// TIA Portal V17 export
// export: Created 2022-07-20T06:59:51.1083772Z, ExportSetting WithDefaults, DisplayName Totally Integrated Automation Portal, DisplayVersion V17, DisplayName TIA Portal Openness, DisplayVersion V17, DisplayName TIA Portal Version Control Interface, DisplayVersion V17, DisplayName SINAMICS Startdrive Advanced, DisplayVersion V17, DisplayName SINAMICS Startdrive G130, G150, S120, S150, SINAMICS MV, S210, DisplayVersion V17, DisplayName SINAMICS Startdrive G110M, G120, G120C, G120D, G120P, G115D, DisplayVersion V17, DisplayName STEP 7 Professional, DisplayVersion V17, DisplayName STEP 7 Safety, DisplayVersion V17, DisplayName WinCC Advanced, DisplayVersion V17
FUNCTION_BLOCK "FB10065_IperPurgeInkCircuit"   // FB10065, LAD
{ S7_Optimized_Access := 'TRUE' }
VERSION : 0.1
// stored: AutoNumber false, IsIECCheckEnabled false, IsRetainMemResEnabled false, MemoryReserve 100, SetENOAutomatically false, UDAEnableTagReadback false
   VAR_INPUT
      PurgeTrayVarnishSensor_1 : Bool;
      PurgeTrayVarnishSensor_2 : Bool;
      Purge1WeighScale_RawWeight : Int;
      Purge1WeighScale_CalibrationWeight_1 : Real;
      Purge1WeighScale_CalibrationWeight_2 : Real;
      Purge1WeighScale_LowWarningThreshold : Real;
      Purge1WeighScale_HighWarningThreshold : Real;
      Purge1WeighScale_LowErrorThreshold : Real;
      Purge1WeighScale_HighErrorThreshold : Real;
      Purge2WeighScale_RawWeight : Int;
      Purge2WeighScale_CalibrationWeight_1 : Real;
      Purge2WeighScale_CalibrationWeight_2 : Real;
      Purge2WeighScale_LowWarningThreshold : Real;
      Purge2WeighScale_HighWarningThreshold : Real;
      Purge2WeighScale_LowErrorThreshold : Real;
      Purge2WeighScale_HighErrorThreshold : Real;
      DrainPurgeTrayTime : Time;
      RequestDrainPurgeTrays : Bool;
   END_VAR
   VAR_OUTPUT
      ActivePurgeOutPump_1 : Bool;
      ActivePurgeOutSolenoidValve_1 : Bool;
      ActivePurgeOutPump_2 : Bool;
      ActivePurgeOutSolenoidValve_2 : Bool;
      Purge1WeighScale_CalibrationStatus_1 : Bool;
      Purge1WeighScale_CalibrationStatus_2 : Bool;
      Purge1WeighScale_LowWarningThresholdReached : Bool;
      Purge1WeighScale_HighWarningThresholdReached : Bool;
      Purge1WeighScale_LowErrorThresholdReached : Bool;
      Purge1WeighScale_HighErrorThresholdReached : Bool;
      Purge1WeighScale_NetWeight : Real;
      "Purge1WeighScale_NetWeight_%" : Real;
      Purge1WeighScale_SensorCalibrated : Bool;
      Purge2WeighScale_CalibrationStatus_1 : Bool;
      Purge2WeighScale_CalibrationStatus_2 : Bool;
      Purge2WeighScale_LowWarningThresholdReached : Bool;
      Purge2WeighScale_HighWarningThresholdReached : Bool;
      Purge2WeighScale_LowErrorThresholdReached : Bool;
      Purge2WeighScale_HighErrorThresholdReached : Bool;
      Purge2WeighScale_NetWeight : Real;
      "Purge2WeighScale_NetWeight_%" : Real;
      Purge2WeighScale_SensorCalibrated : Bool;
      DrainPurgeTraysDone : Bool;
   END_VAR
   VAR_IN_OUT
      Purge1WeighScale_CalibrationDataX_1 : Real;
      Purge1WeighScale_CalibrationDataY_1 : Real;
      Purge1WeighScale_CalibrationDataX_2 : Real;
      Purge1WeighScale_CalibrationDataY_2 : Real;
      Purge1WeighScale_RequestCalibration_1 : Bool;
      Purge1WeighScale_RequestCalibration_2 : Bool;
      Purge1WeighScale_ResetCalibration : Bool;
      Purge2WeighScale_CalibrationDataX_1 : Real;
      Purge2WeighScale_CalibrationDataY_1 : Real;
      Purge2WeighScale_CalibrationDataX_2 : Real;
      Purge2WeighScale_CalibrationDataY_2 : Real;
      Purge2WeighScale_RequestCalibration_1 : Bool;
      Purge2WeighScale_RequestCalibration_2 : Bool;
      Purge2WeighScale_ResetCalibration : Bool;
   END_VAR
   VAR
      PurgeInkCircuitStateDiagram : Int;
      R_TRIG_RequestDrainPurgeTrays : R_TRIG;
      F_TRIG_RequestDrainPurgeTrays { S7_SetPoint := 'True'} : F_TRIG;
      F_TRIG_PurgeTrayVarnishSensor_1 : F_TRIG;
      F_TRIG_PurgeTrayVarnishSensor_2 : F_TRIG;
      TON_DrainPurgeTray { S7_SetPoint := 'True'} : TON_TIME;
      TON_Safety { S7_SetPoint := 'True'} : TON_TIME;
      FB10030_AnalogicalSensor_TLMScale_PurgeWasteWeighScale_1 { S7_SetPoint := 'True'} : "FB10030_AnalogicalSensor";
      FB10030_AnalogicalSensor_TLMScale_PurgeWasteWeighScale_2 { S7_SetPoint := 'True'} : "FB10030_AnalogicalSensor";
   END_VAR
   VAR CONSTANT
      WAIT_FOR_PURGE_INK_REQUESTS : Int := 0;
      DRAIN_PURGE_TRAY : Int := 20;
      PURGE_INK_REQUESTS_DONE : Int := 30;
   END_VAR
BEGIN

REGION Network 1 (SCL): First Scan
   IF "FirstScan" THEN
       #DrainPurgeTraysDone := FALSE;
   END_IF;
END_REGION

REGION Network 2 (SCL): Edge Signals & Timers
   REGION EDGE SIGNALS
       #R_TRIG_RequestDrainPurgeTrays(CLK := #RequestDrainPurgeTrays);

       #F_TRIG_RequestDrainPurgeTrays(CLK := #RequestDrainPurgeTrays);
       #F_TRIG_PurgeTrayVarnishSensor_1(CLK := #PurgeTrayVarnishSensor_1);
       #F_TRIG_PurgeTrayVarnishSensor_2(CLK := #PurgeTrayVarnishSensor_2);
   END_REGION

   REGION TIMERS
       #TON_DrainPurgeTray(IN := #PurgeInkCircuitStateDiagram = #DRAIN_PURGE_TRAY AND #PurgeTrayVarnishSensor_1 AND #PurgeTrayVarnishSensor_2,
                           PT := #DrainPurgeTrayTime);
       #TON_Safety(IN := #ActivePurgeOutPump_1 AND #ActivePurgeOutPump_2,
                   PT := T#240s);
   END_REGION
END_REGION

REGION Network 3: Purge Out 1 Weigh Scale Management
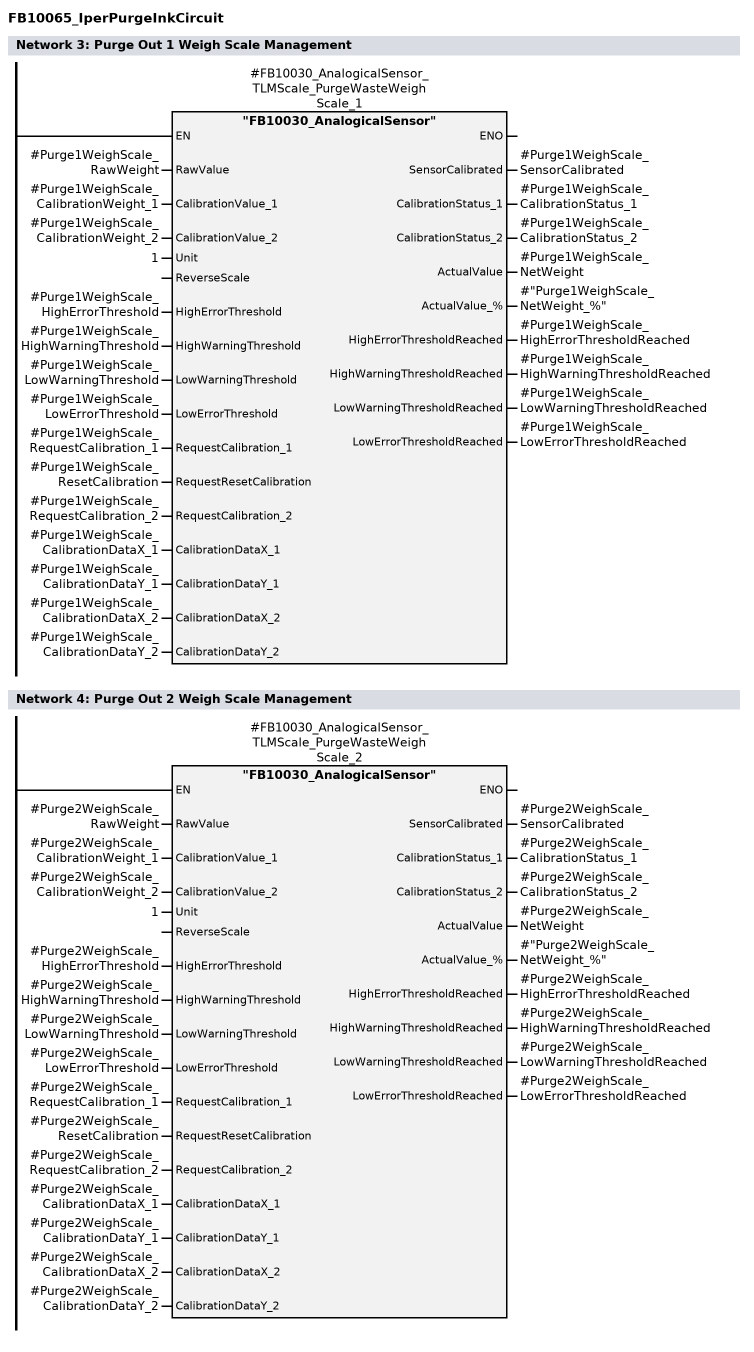
   RUNG wire#powerrail
      #FB10030_AnalogicalSensor_TLMScale_PurgeWasteWeighScale_1(RawValue := #Purge1WeighScale_RawWeight, CalibrationValue_1 := #Purge1WeighScale_CalibrationWeight_1, CalibrationValue_2 := #Purge1WeighScale_CalibrationWeight_2, Unit := 1, ReverseScale :=, HighErrorThreshold := #Purge1WeighScale_HighErrorThreshold, HighWarningThreshold := #Purge1WeighScale_HighWarningThreshold, LowWarningThreshold := #Purge1WeighScale_LowWarningThreshold, LowErrorThreshold := #Purge1WeighScale_LowErrorThreshold, RequestCalibration_1 := #Purge1WeighScale_RequestCalibration_1, RequestResetCalibration := #Purge1WeighScale_ResetCalibration, RequestCalibration_2 := #Purge1WeighScale_RequestCalibration_2, CalibrationDataX_1 := #Purge1WeighScale_CalibrationDataX_1, CalibrationDataY_1 := #Purge1WeighScale_CalibrationDataY_1, CalibrationDataX_2 := #Purge1WeighScale_CalibrationDataX_2, CalibrationDataY_2 := #Purge1WeighScale_CalibrationDataY_2, SensorCalibrated => #Purge1WeighScale_SensorCalibrated, CalibrationStatus_1 => #Purge1WeighScale_CalibrationStatus_1, CalibrationStatus_2 => #Purge1WeighScale_CalibrationStatus_2, ActualValue => #Purge1WeighScale_NetWeight, "ActualValue_%" => #"Purge1WeighScale_NetWeight_%", HighErrorThresholdReached => #Purge1WeighScale_HighErrorThresholdReached, HighWarningThresholdReached => #Purge1WeighScale_HighWarningThresholdReached, LowWarningThresholdReached => #Purge1WeighScale_LowWarningThresholdReached, LowErrorThresholdReached => #Purge1WeighScale_LowErrorThresholdReached)
   END_RUNG
   // the same network as SCL:
   #FB10030_AnalogicalSensor_TLMScale_PurgeWasteWeighScale_1(RawValue := #Purge1WeighScale_RawWeight,   // "FB10030_AnalogicalSensor"
                           CalibrationValue_1 := #Purge1WeighScale_CalibrationWeight_1,
                           CalibrationValue_2 := #Purge1WeighScale_CalibrationWeight_2,
                           Unit := 1,
                           HighErrorThreshold := #Purge1WeighScale_HighErrorThreshold,
                           HighWarningThreshold := #Purge1WeighScale_HighWarningThreshold,
                           LowWarningThreshold := #Purge1WeighScale_LowWarningThreshold,
                           LowErrorThreshold := #Purge1WeighScale_LowErrorThreshold,
                           RequestCalibration_1 := #Purge1WeighScale_RequestCalibration_1,
                           RequestResetCalibration := #Purge1WeighScale_ResetCalibration,
                           RequestCalibration_2 := #Purge1WeighScale_RequestCalibration_2,
                           CalibrationDataX_1 := #Purge1WeighScale_CalibrationDataX_1,
                           CalibrationDataY_1 := #Purge1WeighScale_CalibrationDataY_1,
                           CalibrationDataX_2 := #Purge1WeighScale_CalibrationDataX_2,
                           CalibrationDataY_2 := #Purge1WeighScale_CalibrationDataY_2,
                           SensorCalibrated => #Purge1WeighScale_SensorCalibrated,
                           CalibrationStatus_1 => #Purge1WeighScale_CalibrationStatus_1,
                           CalibrationStatus_2 => #Purge1WeighScale_CalibrationStatus_2,
                           ActualValue => #Purge1WeighScale_NetWeight,
                           "ActualValue_%" => #"Purge1WeighScale_NetWeight_%",
                           HighErrorThresholdReached => #Purge1WeighScale_HighErrorThresholdReached,
                           HighWarningThresholdReached => #Purge1WeighScale_HighWarningThresholdReached,
                           LowWarningThresholdReached => #Purge1WeighScale_LowWarningThresholdReached,
                           LowErrorThresholdReached => #Purge1WeighScale_LowErrorThresholdReached);
END_REGION

REGION Network 4: Purge Out 2 Weigh Scale Management
   RUNG wire#powerrail
      #FB10030_AnalogicalSensor_TLMScale_PurgeWasteWeighScale_2(RawValue := #Purge2WeighScale_RawWeight, CalibrationValue_1 := #Purge2WeighScale_CalibrationWeight_1, CalibrationValue_2 := #Purge2WeighScale_CalibrationWeight_2, Unit := 1, ReverseScale :=, HighErrorThreshold := #Purge2WeighScale_HighErrorThreshold, HighWarningThreshold := #Purge2WeighScale_HighWarningThreshold, LowWarningThreshold := #Purge2WeighScale_LowWarningThreshold, LowErrorThreshold := #Purge2WeighScale_LowErrorThreshold, RequestCalibration_1 := #Purge2WeighScale_RequestCalibration_1, RequestCalibration_2 := #Purge2WeighScale_RequestCalibration_2, RequestResetCalibration := #Purge2WeighScale_ResetCalibration, CalibrationDataX_1 := #Purge2WeighScale_CalibrationDataX_1, CalibrationDataY_1 := #Purge2WeighScale_CalibrationDataY_1, CalibrationDataX_2 := #Purge2WeighScale_CalibrationDataX_2, CalibrationDataY_2 := #Purge2WeighScale_CalibrationDataY_2, SensorCalibrated => #Purge2WeighScale_SensorCalibrated, CalibrationStatus_1 => #Purge2WeighScale_CalibrationStatus_1, CalibrationStatus_2 => #Purge2WeighScale_CalibrationStatus_2, ActualValue => #Purge2WeighScale_NetWeight, "ActualValue_%" => #"Purge2WeighScale_NetWeight_%", HighErrorThresholdReached => #Purge2WeighScale_HighErrorThresholdReached, HighWarningThresholdReached => #Purge2WeighScale_HighWarningThresholdReached, LowWarningThresholdReached => #Purge2WeighScale_LowWarningThresholdReached, LowErrorThresholdReached => #Purge2WeighScale_LowErrorThresholdReached)
   END_RUNG
   // the same network as SCL:
   #FB10030_AnalogicalSensor_TLMScale_PurgeWasteWeighScale_2(RawValue := #Purge2WeighScale_RawWeight,   // "FB10030_AnalogicalSensor"
                           CalibrationValue_1 := #Purge2WeighScale_CalibrationWeight_1,
                           CalibrationValue_2 := #Purge2WeighScale_CalibrationWeight_2,
                           Unit := 1,
                           HighErrorThreshold := #Purge2WeighScale_HighErrorThreshold,
                           HighWarningThreshold := #Purge2WeighScale_HighWarningThreshold,
                           LowWarningThreshold := #Purge2WeighScale_LowWarningThreshold,
                           LowErrorThreshold := #Purge2WeighScale_LowErrorThreshold,
                           RequestCalibration_1 := #Purge2WeighScale_RequestCalibration_1,
                           RequestResetCalibration := #Purge2WeighScale_ResetCalibration,
                           RequestCalibration_2 := #Purge2WeighScale_RequestCalibration_2,
                           CalibrationDataX_1 := #Purge2WeighScale_CalibrationDataX_1,
                           CalibrationDataY_1 := #Purge2WeighScale_CalibrationDataY_1,
                           CalibrationDataX_2 := #Purge2WeighScale_CalibrationDataX_2,
                           CalibrationDataY_2 := #Purge2WeighScale_CalibrationDataY_2,
                           SensorCalibrated => #Purge2WeighScale_SensorCalibrated,
                           CalibrationStatus_1 => #Purge2WeighScale_CalibrationStatus_1,
                           CalibrationStatus_2 => #Purge2WeighScale_CalibrationStatus_2,
                           ActualValue => #Purge2WeighScale_NetWeight,
                           "ActualValue_%" => #"Purge2WeighScale_NetWeight_%",
                           HighErrorThresholdReached => #Purge2WeighScale_HighErrorThresholdReached,
                           HighWarningThresholdReached => #Purge2WeighScale_HighWarningThresholdReached,
                           LowWarningThresholdReached => #Purge2WeighScale_LowWarningThresholdReached,
                           LowErrorThresholdReached => #Purge2WeighScale_LowErrorThresholdReached);
END_REGION

REGION Network 5 (SCL): Purge Ink Circuit Management
   CASE #PurgeInkCircuitStateDiagram OF
       #WAIT_FOR_PURGE_INK_REQUESTS:
           IF #R_TRIG_RequestDrainPurgeTrays.Q OR #F_TRIG_PurgeTrayVarnishSensor_1.Q OR #F_TRIG_PurgeTrayVarnishSensor_2.Q THEN
               #DrainPurgeTraysDone := FALSE;
               #PurgeInkCircuitStateDiagram := #DRAIN_PURGE_TRAY;
           END_IF;
       #DRAIN_PURGE_TRAY:
           #ActivePurgeOutSolenoidValve_1 := TRUE;
           #ActivePurgeOutSolenoidValve_2 := TRUE;
           #ActivePurgeOutPump_2 := TRUE;
           #ActivePurgeOutPump_1 := TRUE;
           IF (#PurgeTrayVarnishSensor_1 AND #PurgeTrayVarnishSensor_2 AND #TON_DrainPurgeTray.Q) OR #F_TRIG_RequestDrainPurgeTrays.Q OR #TON_Safety.Q THEN
               #ActivePurgeOutSolenoidValve_1 := FALSE;
               #ActivePurgeOutSolenoidValve_2 := FALSE;
               #ActivePurgeOutPump_2 := FALSE;
               #ActivePurgeOutPump_1 := FALSE;
               #DrainPurgeTraysDone := TRUE;
               #PurgeInkCircuitStateDiagram := #PURGE_INK_REQUESTS_DONE;
           END_IF;
       #PURGE_INK_REQUESTS_DONE:
           #PurgeInkCircuitStateDiagram := #WAIT_FOR_PURGE_INK_REQUESTS;
   END_CASE;
END_REGION
END_FUNCTION_BLOCK
